// TIA Portal V17 export
// export: Created 2024-01-30T08:49:10.1779437Z, ExportSetting WithDefaults, DisplayName Totally Integrated Automation Portal, DisplayVersion V17 Update 6, DisplayName TIA Portal Openness, DisplayVersion V17 Update 6, DisplayName TIA Portal Version Control Interface, DisplayVersion V17, DisplayName STEP 7 Professional, DisplayVersion V17 Update 6, DisplayName STEP 7 Safety, DisplayVersion V17 Update 6, DisplayName WinCC Advanced, DisplayVersion V17 Update 6
ORGANIZATION_BLOCK "Main"   // OB1, LAD, ProgramCycle
TITLE = "Main Program Sweep (Cycle)"
{ S7_Optimized_Access := 'TRUE' }
VERSION : 0.1
// stored: AutoNumber true, IsIECCheckEnabled false, SetENOAutomatically false
   VAR_INPUT
      Initial_Call : Bool;   // Initial call of this OB
      Remanence : Bool;   // =True, if remanent data are available
   END_VAR
   VAR_TEMP
      RetVAl : Int;
   END_VAR
BEGIN

REGION Network 1: Read Local Time
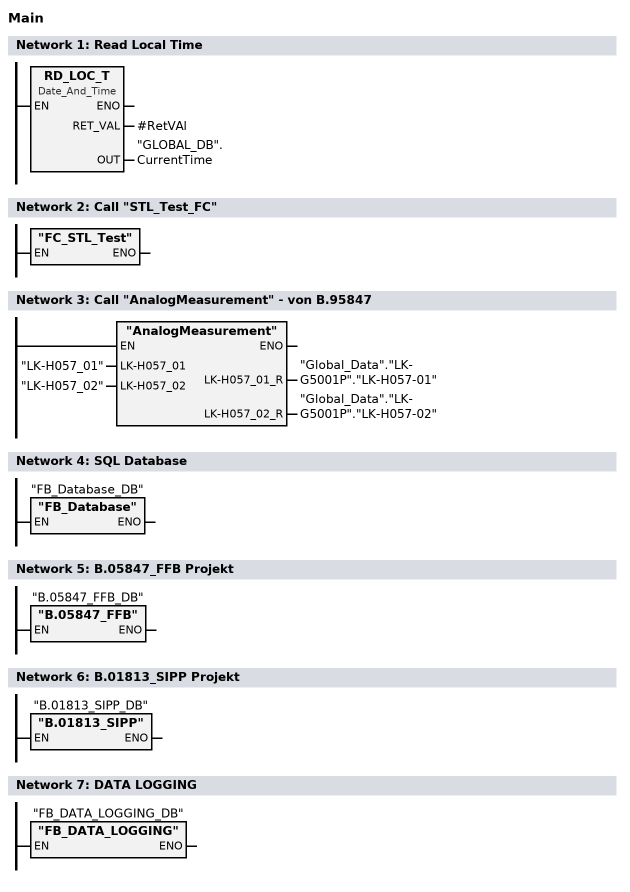
   RUNG wire#powerrail
      { S7_Templates := "date_type := Date_And_Time" } RD_LOC_T(RET_VAL => #RetVAl, OUT => "GLOBAL_DB".CurrentTime)
   END_RUNG
   // the same network as SCL:
   #RetVAl := RD_LOC_T(OUT => "GLOBAL_DB".CurrentTime);
END_REGION

REGION Network 2: Call "STL_Test_FC"
   RUNG wire#powerrail
      "FC_STL_Test"()
   END_RUNG
   // the same network as SCL:
   "FC_STL_Test"();
END_REGION

REGION Network 3: Call "AnalogMeasurement" - von B.95847
   RUNG wire#powerrail
      "AnalogMeasurement"("LK-H057_01" := "LK-H057_01", "LK-H057_02" := "LK-H057_02", "LK-H057_01_R" => "Global_Data"."LK-G5001P"."LK-H057-01", "LK-H057_02_R" => "Global_Data"."LK-G5001P"."LK-H057-02")
   END_RUNG
   // the same network as SCL:
   "AnalogMeasurement"("LK-H057_01" := "LK-H057_01",
                       "LK-H057_02" := "LK-H057_02",
                       "LK-H057_01_R" => "Global_Data"."LK-G5001P"."LK-H057-01",
                       "LK-H057_02_R" => "Global_Data"."LK-G5001P"."LK-H057-02");
END_REGION

REGION Network 4: SQL Database
   RUNG wire#powerrail
      "FB_Database_DB"()
   END_RUNG
   // the same network as SCL:
   "FB_Database_DB"();   // "FB_Database"
END_REGION

REGION Network 5: B.05847_FFB Projekt
   RUNG wire#powerrail
      "B.05847_FFB_DB"()
   END_RUNG
   // the same network as SCL:
   "B.05847_FFB_DB"();   // "B.05847_FFB"
END_REGION

REGION Network 6: B.01813_SIPP Projekt
   RUNG wire#powerrail
      "B.01813_SIPP_DB"()
   END_RUNG
   // the same network as SCL:
   "B.01813_SIPP_DB"();   // "B.01813_SIPP"
END_REGION

REGION Network 7: DATA LOGGING
   RUNG wire#powerrail
      "FB_DATA_LOGGING_DB"()
   END_RUNG
   // the same network as SCL:
   "FB_DATA_LOGGING_DB"();   // "FB_DATA_LOGGING"
END_REGION
END_ORGANIZATION_BLOCK
